(* PLC project Sin nombre, Desconocido Sin nombre 1 *)
(* stored: creationDateTime 2024-10-26T19:00:37, modificationDateTime 2024-10-27T01:21:52 *)

PROGRAM program0
  VAR
    TON2 : TON;
    TP2 : TP;
    TP3 : TP;
    TOF1 : TOF;
    timer : BOOL := 1;
    luz_1 : BOOL := 0;
    luz_2 : BOOL := 0;
    probar_sig : BOOL := 0;
    acumular : BOOL := 0;
    timer_corrido : BOOL := 0;
  END_VAR
  VAR
    sensor AT %IW0.0 : UINT := 0;
    acum AT %MW0.0 : UINT := 0;
  END_VAR
  VAR
    actual : INT := 3;
    tope_normal : UINT := 0;  (* modificar este y el de abajo *)
    tope_alto : UINT := 0;
  END_VAR
  VAR  (* added by the conversion: wires and edge detectors of the diagram *)
    _EQ79_ENO : BOOL;
    _EQ79_OUT : BOOL;
    _LT41_ENO : BOOL;
    _LT41_OUT : BOOL;
    _GE83_ENO : BOOL;
    _GE83_OUT : BOOL;
    _EQ32_ENO : BOOL;
    _EQ32_OUT : BOOL;
    _LT97_ENO : BOOL;
    _LT97_OUT : BOOL;
    _GE55_ENO : BOOL;
    _GE55_OUT : BOOL;
    _ADD67_ENO : BOOL;
    _ADD67_OUT : UINT;
  END_VAR

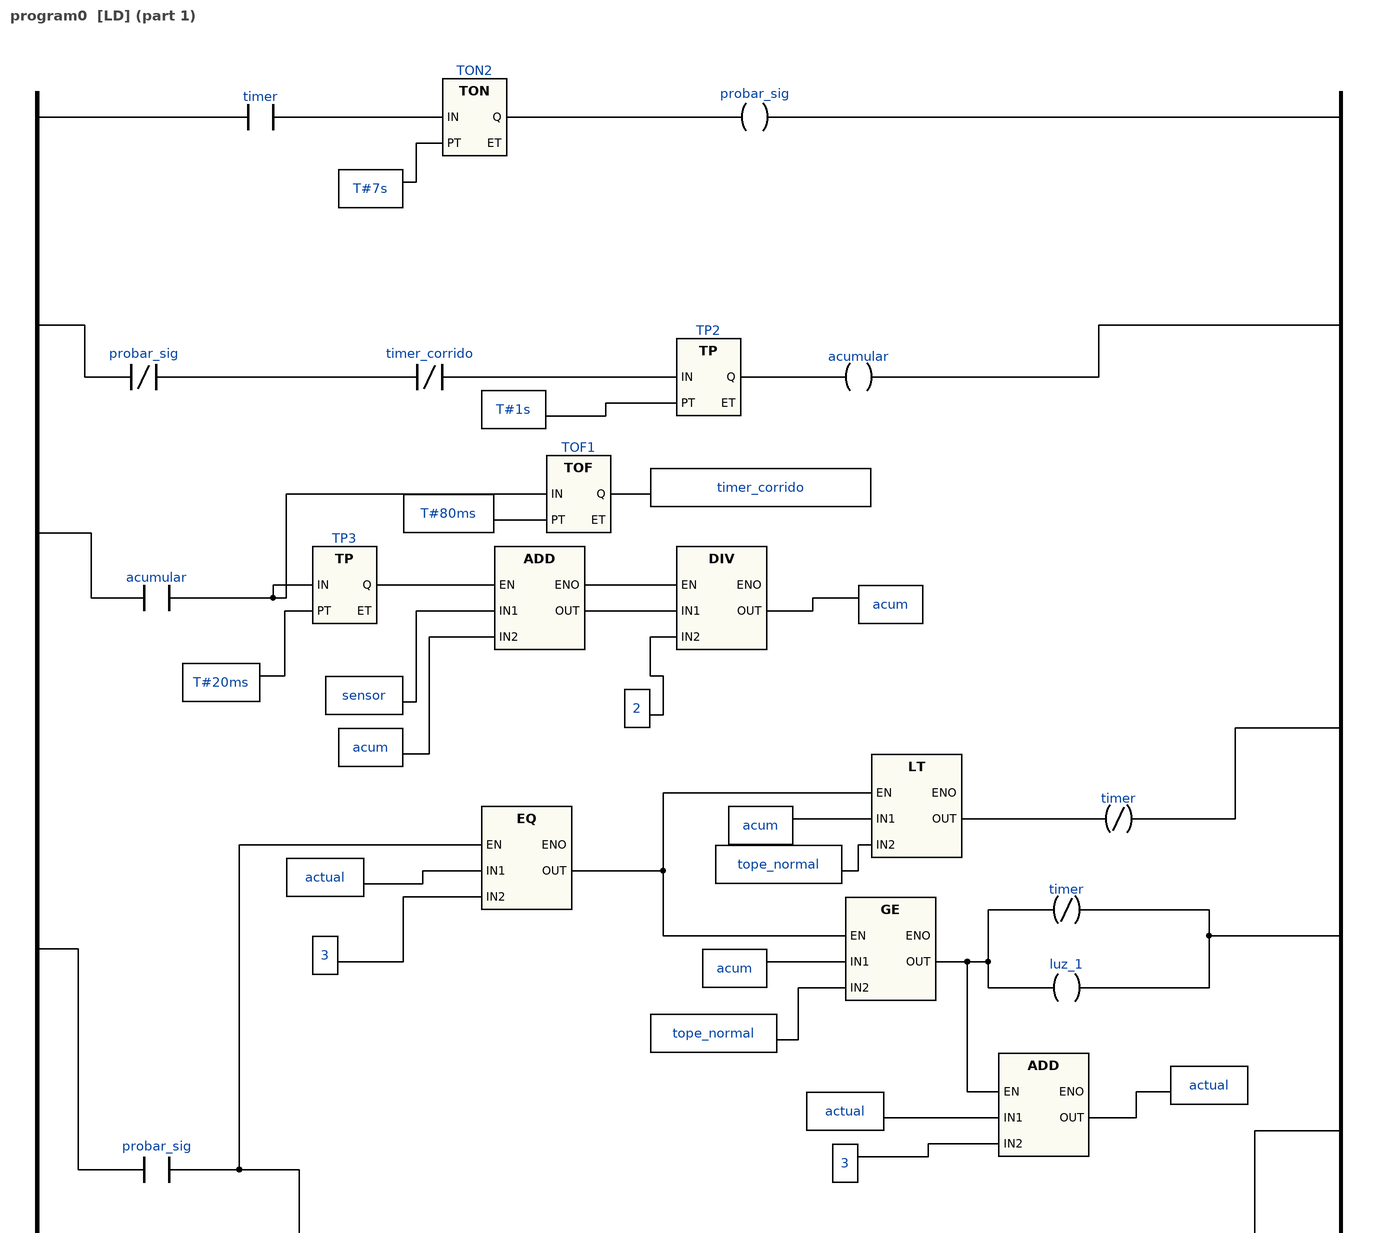
(* LD diagram, written out as Structured Text *)
TON2(IN := timer, PT := T#7s);
probar_sig := TON2.Q;
TP2(IN := NOT probar_sig AND NOT timer_corrido, PT := T#1s);
acumular := TP2.Q;
_EQ79_OUT := EQ(EN := probar_sig, IN1 := actual, IN2 := 3, ENO => _EQ79_ENO);
_LT41_OUT := LT(EN := _EQ79_OUT, IN1 := acum, IN2 := tope_normal, ENO => _LT41_ENO);
timer := NOT _LT41_OUT;
_GE83_OUT := GE(EN := _EQ79_OUT, IN1 := acum, IN2 := tope_normal, ENO => _GE83_ENO);
timer := NOT _GE83_OUT;
luz_1 := _GE83_OUT;
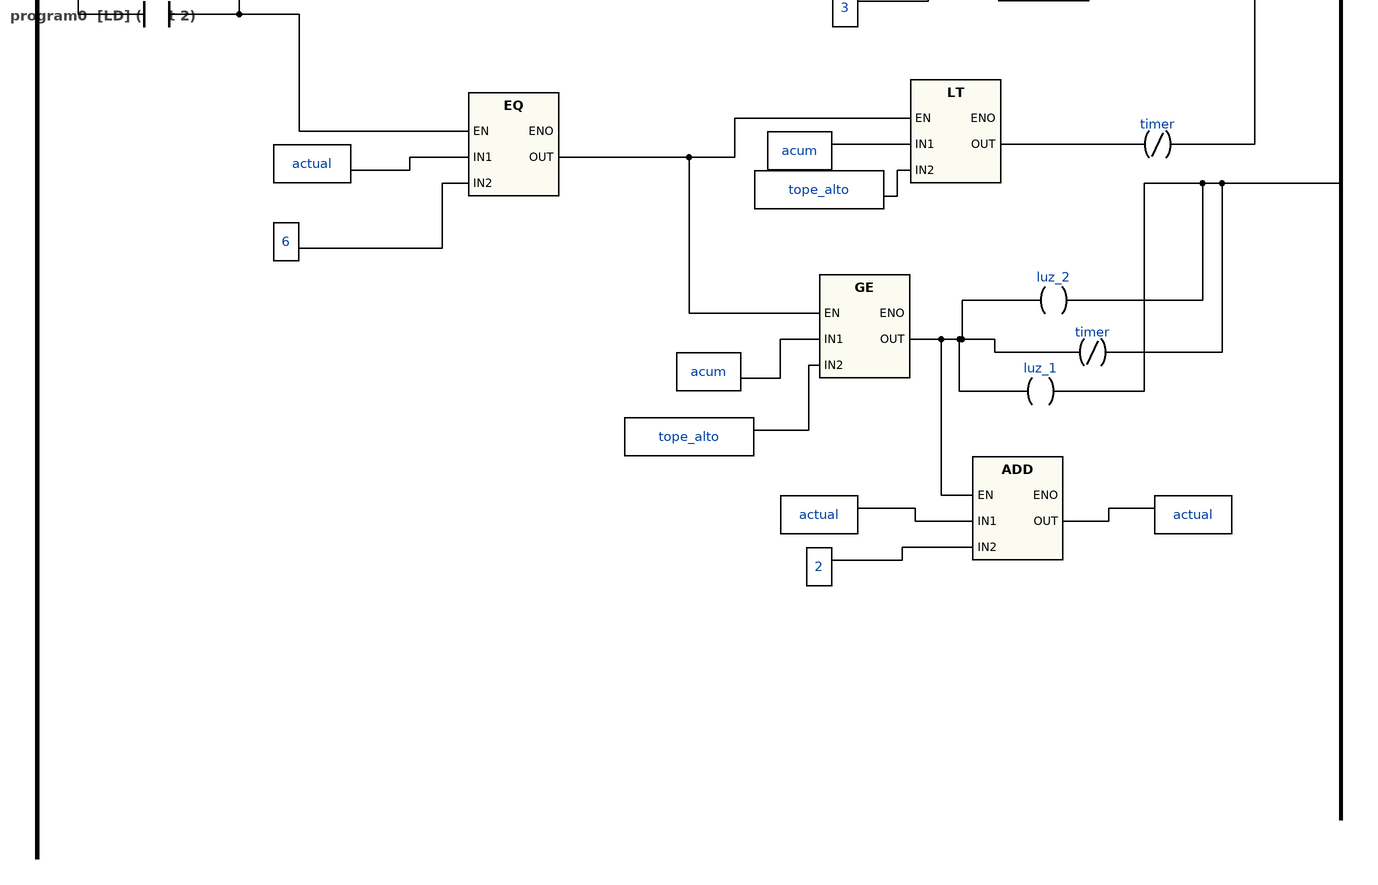
_EQ32_OUT := EQ(EN := probar_sig, IN1 := actual, IN2 := 6, ENO => _EQ32_ENO);
_LT97_OUT := LT(EN := _EQ32_OUT, IN1 := acum, IN2 := tope_alto, ENO => _LT97_ENO);
timer := NOT _LT97_OUT;
_GE55_OUT := GE(EN := _EQ32_OUT, IN1 := acum, IN2 := tope_alto, ENO => _GE55_ENO);
luz_2 := _GE55_OUT;
luz_1 := _GE55_OUT;
TP3(IN := acumular, PT := T#20ms);
_ADD67_OUT := ADD(EN := TP3.Q, IN1 := sensor, IN2 := acum, ENO => _ADD67_ENO);
IF _ADD67_ENO THEN acum := _ADD67_OUT / 2; END_IF;
TOF1(IN := acumular, PT := T#80ms);
timer_corrido := TOF1.Q;
timer := NOT _GE55_OUT;
IF _GE83_OUT THEN actual := actual + 3; END_IF;
IF _GE55_OUT THEN actual := actual + 2; END_IF;
END_PROGRAM

CONFIGURATION Config0
  RESOURCE Res0 ON PLC
    TASK task0(INTERVAL := T#20ms, PRIORITY := 0);
  END_RESOURCE
END_CONFIGURATION
